SYSTEM System (* System Configuration *)
  (* Version 0.0, 2/18/2025, SESA575785, Schneider Electric *)
  APPLICATION APP1
  END_APPLICATION
  DEVICE EcoRT_0 : Soft_dPAC
    RESOURCE RES0 : EMB_RES_ECO
    END_RESOURCE
  END_DEVICE
END_SYSTEM
(* other elements stored in the file *)
(* DefaultLayer Name=Default *)
